// Mitsubishi GX Works2 project: PID_master_Q00_26_04_2021   PLC: Q00

// global labels: Global1
VAR_GLOBAL
  Input_ManualMode AT M500 : BOOL;  (* Valg av Manuell "1" eller Auto "0" *)
  Input_OperationModus AT M501 : BOOL;  (* Valg av direkte "1" eller Revers "0" Regulering *)
  Input_IntegratorModus AT M502 : BOOL;  (* Valg av Integrator virkning på regulator *)
  Input_DerivatorModus AT M503 : BOOL;  (* Valg av Derivator virkning på regulator *)
  Input_SamplingsTime AT D200 : INT;  (* Samplingstid sendt til PID *)
  Input_Referance AT D204 : INT;  (* Referanse verdi sendt til PID *)
  Input_ManualValue AT D208 : INT;  (* Manuell verdi sendt til PID *)
  Input_NomValue AT D210 : INT;  (* Nominelt pådrag *)
  Input_MaxPådrag AT D212 : INT;  (* Max pådrag *)
  Input_MinPådrag AT D214 : INT;  (* Min pådrag *)
  Input_KpValue AT D218 : INT;  (* Valg av Kp verdi *)
  Input_TiValue AT D220 : INT;  (* Valge av Ti verdi *)
  Input_TdValue AT D222 : INT;  (* Valg av Td verdi *)
  Input_NValue AT D224 : INT;  (* Valg av N verdi *)
  Input_TtValue AT D226 : INT;  (* Valg av Tt verdi *)
  Input_FF_TtValue AT D228 : INT;  (* Valg av Tt verdi til LeadLag blokk *)
  Input_FF_TnValue AT D230 : INT;  (* Valg av Tn verdi til LeadLag blokk *)
  Input_FF_KLLValue AT D232 : INT;  (* Valg av KLL verdi til LeadLag blokk *)
  Input_ErrorValue AT D238 : INT;  (* Beregnet avvik *)
  Pump AT M400 : BOOL;  (* Kontaktor til drift av pumpe *)
  AlarmLamp AT M401 : BOOL;  (* Alarm lampe til systemet *)
  MagnetValve_1 AT M404 : BOOL;  (* Magnetventil 1 *)
  MagnetValve_2 AT M405 : BOOL;  (* Magnetventil 2 *)
  MagnetValve_3 AT M406 : BOOL;  (* Magnetventil 3 *)
  Input_Pump AT M504 : BOOL;  (* Start signal til pumpe fra Master *)
  Input_AlarmLamp AT M505 : BOOL;  (* Start signal til Alarm lampe fra Master *)
  Input_MagnetValve_1 AT M506 : BOOL;  (* Start signal til Magnetventil 1 fra Master *)
  Input_MagnetValve_2 AT M507 : BOOL;  (* Start signal til Magnetventil 2 fra Master *)
  Input_MagnetValve_3 AT M508 : BOOL;  (* Start signal til Magnetventil 3 fra Master *)
  Input_Flow AT D240 : INT;  (* Scaled and converted Flow signal in percentage. *)
  Output_Total AT D236 : INT;  (* Totalt utgangsignal summert *)
  Input_Process AT D206 : INT;  (* Prosess verdi Sendt til PID *)
  Output_Tank_high AT M600 : BOOL;
  Output_Tank_low AT M601 : BOOL;
  Output_Tank_high_high AT M602 : BOOL;
  Output_Tank_low_low AT M603 : BOOL;
  Output_Normal_ErrorSignal AT M604 : BOOL;
  Output_Critical_ErrorSignal AT M605 : BOOL;
  Output_Power_failure AT M606 : BOOL;
  Input_Acknowledge_normalHigh AT M608 : BOOL;
  Input_Acknowledge_normalLow AT M609 : BOOL;
  Input_Acknowledge_criticalHigh AT M610 : BOOL;
  Input_Acknowledge_criticalLow AT M611 : BOOL;
  Input_Acknowledge_powerFailure AT M612 : BOOL;
  Input_Acknowledge_Normal_Error AT M613 : BOOL;
  Input_Acknowledge_Critical_Error AT M614 : BOOL;
  Input_PID_ON AT M509 : BOOL;  (* On Off switch for PID Function block *)
  Input_LeadLag1_ON AT M510 : BOOL;  (* On Off switch for Leadlag function block1 *)
  Input_LeadLag2_ON AT M511 : BOOL;  (* On Off switch for Leadlag function block 2 *)
  Communication_trouble_detection AT X1 : BOOL;
  Input_Acknowledge_profibus_error AT M641 : BOOL;
  Master_Acknowledge_powerFailure AT M644 : BOOL;
  Output_Profibus_error_signal AT M512 : BOOL;
  Master_Power_failure AT M513 : BOOL;
  Intouch_Acknowledge_normalLow AT M408 : BOOL;
  Intouch_Acknowledge_criticalHigh AT M409 : BOOL;
  Intouch_Acknowledge_criticalLow AT M410 : BOOL;
  Intouch_Acknowledge_Slave_Power AT M411 : BOOL;
  Intouch_Acknowledge_Normal_Error AT M412 : BOOL;
  Intouch_Acknowledge_Crit_Error AT M413 : BOOL;
  Intouch_Acknowledge_prof_error AT M414 : BOOL;
  Intouch_Acknowledge_Master_Power AT M415 : BOOL;
  Intouch_Acknowledge_normalHigh AT M416 : BOOL;
  Intouch_Alarm_normalLow AT D417 : INT;
  Intouch_Alarm_normalHigh AT D418 : INT;
  Intouch_Alarm_criticalLow AT D419 : INT;
  Intouch_Alarm_criticalHigh AT D420 : INT;
  Intouch_Alarm_SlavePower AT D421 : INT;
  Intouch_Alarm_MasterPower AT D422 : INT;
  Intouch_Alarm_NormalError AT D423 : INT;
  Intouch_Alarm_CriticalError AT D424 : INT;
  Intouch_Alarm_ProfError AT D425 : INT;
END_VAR

PROGRAM POU_01
(* structured ladder/FBD written out as ST: instructions are called as NAME(EN, inputs, outputs); _pN, _eN, _tN stand for wires *)
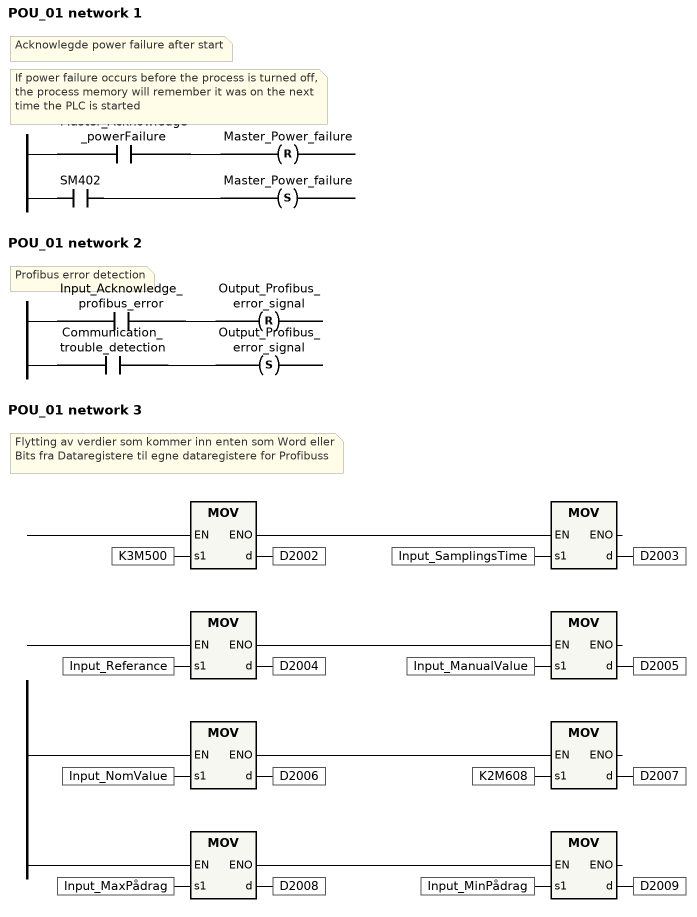
(* network 1 *)
(* Acknowlegde power failure after start *)
(* If power failure occurs before the process is turned off, the process memory will remember it was on the next time the PLC is started *)
RST(Master_Acknowledge_powerFailure, Master_Power_failure);
SET(SM402, Master_Power_failure);
(* network 2 *)
(* Profibus error detection *)
RST(Input_Acknowledge_profibus_error, Output_Profibus_error_signal);
SET(Communication_trouble_detection, Output_Profibus_error_signal);
(* network 3 *)
(* Flytting av verdier som kommer inn enten som Word eller Bits fra Dataregistere til egne dataregistere for Profibuss *)
_e1 := MOV(TRUE, K3M500, D2002);
MOV(_e1, Input_SamplingsTime, D2003);
_e2 := MOV(TRUE, Input_Referance, D2004);
MOV(_e2, Input_ManualValue, D2005);
_e3 := MOV(TRUE, Input_NomValue, D2006);
MOV(_e3, K2M608, D2007);
_e4 := MOV(TRUE, Input_MaxPådrag, D2008);
MOV(_e4, Input_MinPådrag, D2009);
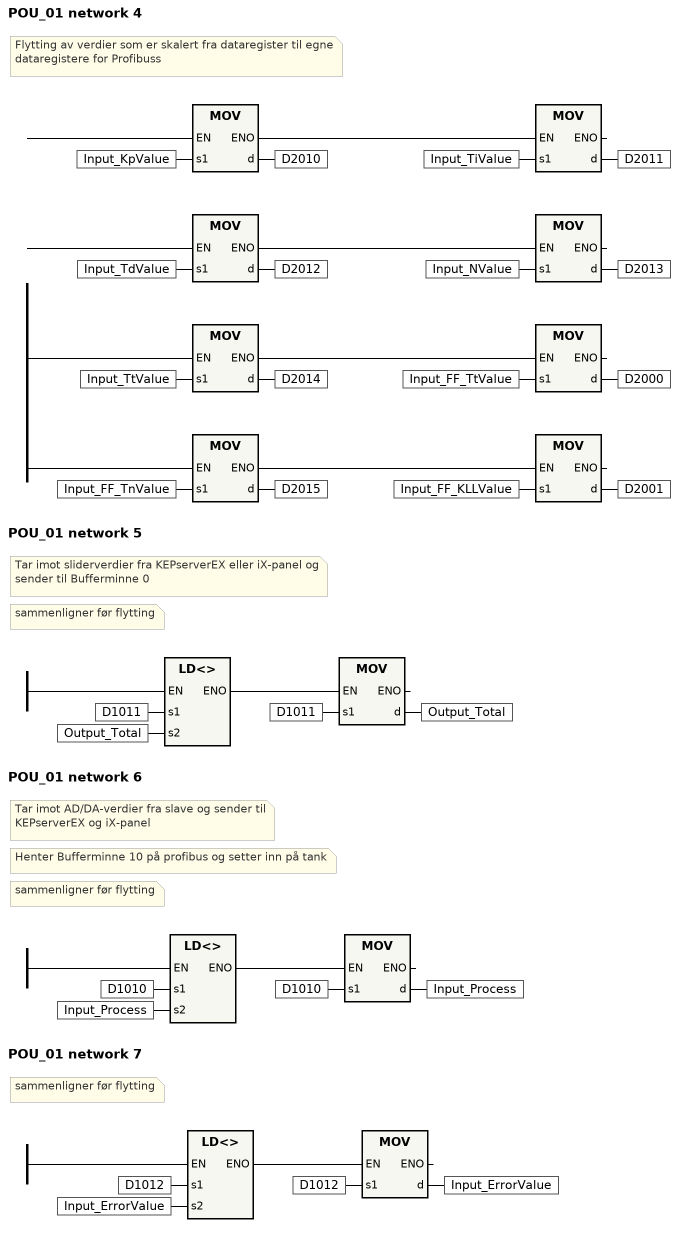
(* network 4 *)
(* Flytting av verdier som er skalert fra dataregister til egne dataregistere for Profibuss *)
_e1 := MOV(TRUE, Input_KpValue, D2010);
MOV(_e1, Input_TiValue, D2011);
_e2 := MOV(TRUE, Input_TdValue, D2012);
MOV(_e2, Input_NValue, D2013);
_e3 := MOV(TRUE, Input_TtValue, D2014);
MOV(_e3, Input_FF_TtValue, D2000);
_e4 := MOV(TRUE, Input_FF_TnValue, D2015);
MOV(_e4, Input_FF_KLLValue, D2001);
(* network 5 *)
(* Tar imot sliderverdier fra KEPserverEX eller iX-panel og sender til Bufferminne 0 *)
(* sammenligner før flytting *)
_e1 := LD<>(TRUE, D1011, Output_Total);
MOV(_e1, D1011, Output_Total);
(* network 6 *)
(* Tar imot AD/DA-verdier fra slave og sender til KEPserverEX og iX-panel *)
(* Henter Bufferminne 10 på profibus og setter inn på tank *)
(* sammenligner før flytting *)
_e1 := LD<>(TRUE, D1010, Input_Process);
MOV(_e1, D1010, Input_Process);
(* network 7 *)
(* sammenligner før flytting *)
_e1 := LD<>(TRUE, D1012, Input_ErrorValue);
MOV(_e1, D1012, Input_ErrorValue);
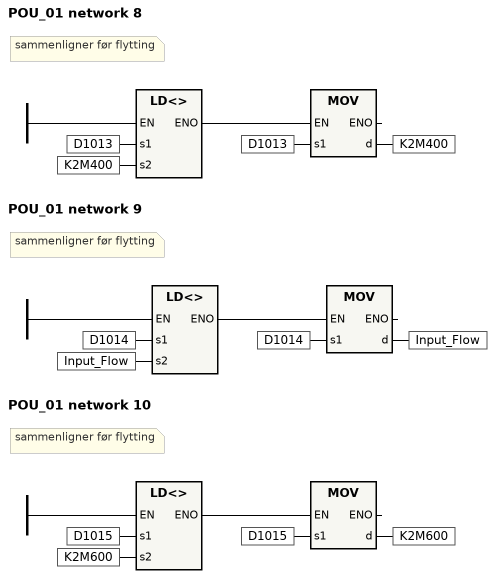
(* network 8 *)
(* sammenligner før flytting *)
_e1 := LD<>(TRUE, D1013, K2M400);
MOV(_e1, D1013, K2M400);
(* network 9 *)
(* sammenligner før flytting *)
_e1 := LD<>(TRUE, D1014, Input_Flow);
MOV(_e1, D1014, Input_Flow);
(* network 10 *)
(* sammenligner før flytting *)
_e1 := LD<>(TRUE, D1015, K2M600);
MOV(_e1, D1015, K2M600);
END_PROGRAM
